(* CODESYS project sql.project
   Title: sql
   Version: 0.0.0.0
   Author: gusta

Project tree, tasks and I/O mapping:
  MyController : TM241CEC24T/U, Schneider Electric, order no. TM241CEC24T/U, version 4.0.6.18
    application Application
      libraries: Standard64, 3.5.2.0 (System); SqlRemoteAccess, 1.0.10.0 (Schneider Electric)
      task MAST (cyclic, interval 2 ms, priority 15) calls POU
      global variables GVL
      program POU [ST]
    DI : Digital Inputs, Schneider Electric, version 4.0.6.18
        input  iwDI_IW0 : WORD  // IW0
        input  ibDI_IB1 : BYTE  // IB1
    DQ : Digital Outputs, Schneider Electric, version 4.0.6.18
        output qwDQ_QW0 : WORD  // QW0
        output qbDQ_QB1 : BYTE  // QB1
    Counters : Counters, Schneider Electric, version 4.0.6.18
    Pulse_Generators : Pulse Generators, Schneider Electric, version 4.0.6.18
    Cartridge_1 : Cartridge, Schneider Electric, version 4.0.6.18
    IO_Bus : IO bus - TM3, Schneider Electric, version 4.0.6.18
      Module_1 : TM3AQ4/G, Schneider Electric, order no. TM3AQ4/G, version 1.0.0.12
          output qiModule_1_QW0 : INT  // QW0
          output qiModule_1_QW1 : INT  // QW1
          output qiModule_1_QW2 : INT  // QW2
          output qiModule_1_QW3 : INT  // QW3
          input  ibModule_1_IBStatusQW0 : BYTE  // IBStatusQW0
          input  ibModule_1_IBStatusQW1 : BYTE  // IBStatusQW1
          input  ibModule_1_IBStatusQW2 : BYTE  // IBStatusQW2
          input  ibModule_1_IBStatusQW3 : BYTE  // IBStatusQW3
      Module_2 : TM3SAF5R/G, Schneider Electric, order no. TM3SAF5R/G, version 1.0.1.12
          input  iwModule_2_IW0 : WORD  // IW0
          output qbModule_2_QB0 : BYTE  // QB0
    COM_Bus : COM bus, Schneider Electric, version 4.0.6.18
    Ethernet_1 : Ethernet Network, Schneider Electric, version 4.0.6.18
    Serial_Line_1 : Serial line, Schneider Electric, version 4.0.6.18
      SoMachine_Network_Manager : SoMachine-Network Manager, Schneider Electric, version 4.0.0.2
    Serial_Line_2 : Serial line, Schneider Electric, version 4.0.6.18
      Modbus_Manager : Modbus Manager, Schneider Electric, version 4.0.0.2
    CAN_1 : CANopen bus, Schneider Electric, version 4.0.6.18
*)

// MyController/Application/GVL
VAR_GLOBAL
END_VAR

// MyController/Application/POU
PROGRAM POU
VAR
	connector: SE_SQL.ST_ConnectionSettings := (wsDbConnectionName := "andreas", wsGwIpAddress := "192.168.1.30", timSqlTimeout := TIME#20s0ms);
	start: BOOL;
	timer: TON;
	String_3: WSTRING(255);
	String_1: WSTRING(255);
	String_2: WSTRING(255);
	
	time_1: INT;
	sql_1: WSTRING(255);
	sql_2: WSTRING(255);
	timer_2: TON;
	state: INT;
	sql: SE_SQL.FB_SqlDbWrite;
	Copy_of_towstringarray: SE_SQL.RequestWstring;
	towstringarray: SE_SQL.RequestWstring;
	My_String: WSTRING(255);
	buffercounter: INT := 0;
	cycle: LINT := 0;
	statementsCounter: INT := 1;
END_VAR


	cycle := cycle + 1;

	String_3 := Standard64.WCONCAT(LINT_TO_WSTRING(cycle*2), ","); // remember to change the cycletime multiplier
	String_1 := Standard64.WCONCAT(String_3 ,DINT_TO_WSTRING(1));
	String_2 := Standard64.WCONCAT(String_1,",");
	My_String := Standard64.WCONCAT(String_2, INT_TO_WSTRING(1));
	towstringarray[1] := Standard64.WCONCAT("INSERT INTO st_logger.test_nr (times, pos, voltage) values(", My_String) ;
	towstringarray[1] := Standard64.WCONCAT(towstringarray[1],");");
	sql(iq_stConnSettings := connector, i_refRequestWstring	:= towstringarray, i_uiNumOfWstrings := 1);
	sql.i_xExecute := TRUE;
	
	IF sql.q_xDone THEN
		sql.i_xExecute := FALSE;
	END_IF

END_PROGRAM
